DATA_BLOCK "DB_Commissioning"
VAR
  str : Array[1..8] of String[60];
  bit : Array[1..8] of Bool;
END_VAR
BEGIN
END_DATA_BLOCK
